Staubli VAL3: getHarmonicMean.pgx

public program getHarmonicMean(num& x_nInput[], num& x_nMean)
  local num l_nCount
  local num l_nSum
begin

  l_nSum = 0

  for l_nCount = 0 to size(x_nInput)-1
    l_nSum = l_nSum + 1/x_nInput[l_nCount]
  endFor

  x_nMean = size(x_nInput)/ l_nSum

end
